{attribute 'linkalways'} 
{attribute 'no_explicit_call' := 'This FB is a CLASS and must be accessed using methods or properties'}
{attribute 'enable_dynamic_creation'}
FUNCTION_BLOCK SequentialSessionIdGenerator Implements I_SessionIdGenerator
VAR
	currentCount : UDINT;
END_VAR

METHOD PUBLIC Generate : T_MAXSTRING
VAR_INPUT
END_VAR
currentCount := currentCount + 1;
Generate := UDINT_TO_STRING(currentCount);
END_METHOD

END_FUNCTION_BLOCK

(* stored: Version 1.1.0.1, ProductVersion 3.1.4024.12
   POU SequentialSessionIdGenerator: Id {1156535e-a90b-0860-3c59-36e2409d0eca}, SpecialFunc None
   Method Generate: Id {2ef8c5f5-ab9c-0cd2-2408-2e410975a162} *)
